(* IEC 61131-3 sources: SIMERLIFT/LOGICAD/SIMERLIFT/src_FBD/BCU/fbdBCU_bess (part 2) *)

  @G(1535) :
     @L(@VF(1532).o, @C(1530).CODE)
    ;
  @G(1536) :
     @L(@VF(1533).o, @C(1530).R)
    ;
  @G(257) :
     @L(@VF(165).o, @C(1).OVTHRES)
    ;
  @G(155) :
     @L(@VF(19).o, @C(1).BAUD)
    ;
  @G(252) :
     @L(@VF(167).o, @C(1).UVTHRES)
    ;
  @G(538) :
     @L(@VF(536).o, @C(1).M_ALL_R)
    ;
  @G(539) :
     @L(@VF(537).o, @C(1).M_AUX_R)
    ;
  @G(206) :
     @L(@VF(24).o, @C(1).N_CELLS)
    ;
  @G(208) :
     @L(@VF(636).o, @C(1).T_CELLS)
    ;
  @G(209) :
     @L(@VF(26).o, @C(1).CHSEL)
    ;
  @G(210) :
     @L(@VF(126).o, @C(1).BRD)
    ;
  @G(213) :
     @L(@VF(235).o, @C(1).CELL)
    ;
  @G(217) :
     @L(@VF(35).o, @C(1).CH)
    ;
  @G(446) :
     @L(@VF(445).o, @C(1).BALV)
    ;
  @G(13) :
     @L(@C(1).VAV, @VF(48).i)
    ;
  @G(11) :
     @L(@C(1).VMINCELL, @VF(30).i)
    ;
  @G(10) :
     @L(@C(1).VMAXCELL, @VF(12).i)
    ;
  @G(8) :
     @L(@C(1).MINCELLBRD, @VF(6).i)
    ;
  @G(3) :
     @L(@C(1).MAXCELLNUM, @VF(5).i)
    ;
  @G(2) :
     @L(@C(1).MAXCELLBRD, @VF(4).i)
    ;
  @G(9) :
     @L(@C(1).MINCELLNUM, @VF(7).i)
    ;
  @G(31) :
     @L(@C(1).VCELL, @VF(18).i)
    ;
  @G(256) :
     @L(@VF(201).o, @C(1).BALENB)
    ;
  @G(41) :
     @L(@C(1).TEMPCELL, @VF(25).i)
    ;
  @G(770) :
     @L(@C(1).VSTACK, @VF(29).i)
    ;
  @G(271) :
     @L(@VF(119).o, @C(1).NTCNOMT_KLV)
    ;
  @G(272) :
     @L(@VF(121).o, @C(1).NTCNOMR_OHM)
    ;
  @G(44) :
     @L(@C(1).BALREG, @VF(72).i)
    ;
  @G(45) :
     @L(@C(1).N_BRD, @VF(154).i)
    ;
  @G(55) :
     @L(@C(1).FAULT, @VF(372).i)
    ;
  @G(128) :
     @L(@C(1).ERR, @VF(654).i)
    ;
  @G(21) :
     @L(@VF(16).o, @C(15).R)
    ;
  @G(27) :
     @L(@VF(20).o, @C(15).CODE)
    ;
  @G(649) :
     @L(@CP(467), @CP(1326)),
     @L(@CP(640), @C(104).CAN_CH),
     @L(@CP(640), @CP(353)),
     @L(@CP(1326), @CP(640)),
     @L(@CP(1326), @C(1004).CAN_CH),
     @L(@VF(638).o, @CP(467)),
     @L(@CP(353), @C(83).CAN_CH),
     @L(@CP(467), @C(136).CAN_CH),
     @L(@CP(353), @C(84).CAN_CH)
    ;
  @G(189) :
     @L(@VF(188).o, @C(1004).CAN_ID)
    ;
  @G(1330) :
     @L(@VF(1120).o, @C(1004).Instant_Current)
    ;
  @G(1331) :
     @L(@VF(1124).o, @C(1004).Selected_BMU_Loc)
    ;
  @G(1332) :
     @L(@VF(1123).o, @C(1004).Selected_Cell_Loc)
    ;
  @G(1333) :
     @L(@VF(1128).o, @C(1004).Cell_Voltage)
    ;
  @G(1334) :
     @L(@VF(1147).o, @C(1004).Cell_Temp)
    ;
  @G(1335) :
     @L(@C(1004).CAN_Error, @VF(1325).i)
    ;
  @G(191) :
     @L(@VF(190).o, @C(104).CAN_ID)
    ;
  @G(1151) :
     @L(@VF(94).o, @C(104).Max_Volt_Cell_Loc)
    ;
  @G(1152) :
     @L(@VF(103).o, @C(104).Max_Volt_BMU_Loc)
    ;
  @G(1153) :
     @L(@VF(105).o, @C(104).Min_Volt_Cell_Loc)
    ;
  @G(1154) :
     @L(@VF(108).o, @C(104).Min_Volt_BMU_Loc)
    ;
  @G(1155) :
     @L(@VF(113).o, @C(104).Average_Cell_Voltage)
    ;
  @G(1156) :
     @L(@VF(114).o, @C(104).Max_Cell_Voltage)
    ;
  @G(1159) :
     @L(@C(104).CAN_Error, @VF(745).i)
    ;
  @G(1160) :
     @L(@VF(115).o, @C(104).Min_Cell_Voltage)
    ;
  @G(782) :
     @L(@C(778).DIV, @VF(779).i)
    ;
  @G(1525) :
     @L(@C(1520).DIV, @VF(1519).i)
    ;
  @G(783) :
     @L(@VF(781).o, @CP(1521)),
     @L(@CP(1521), @C(778).IN2),
     @L(@CP(1521), @C(1520).IN2),
     @L(@CP(1521), @C(1880).IN2),
     @L(@CP(1521), @C(43).IN2)
    ;
  @G(1524) :
     @L(@VF(523).o, @C(1520).IN1)
    ;
  @G(1885) :
     @L(@VF(524).o, @C(1880).IN1)
    ;
  @G(142) :
     @L(@C(466).Overall_Power_kWh, @VF(982).i)
    ;
  @G(717) :
     @L(@C(466).Current_Counter_Ah, @VF(678).i)
    ;
  @G(715) :
     @L(@C(466).Power_kWh, @VF(664).i)
    ;
  @G(713) :
     @L(@C(466).Temp, @VF(663).i)
    ;
  @G(528) :
     @L(@C(466).Voltage3_mV, @VF(525).i)
    ;
  @G(527) :
     @L(@C(466).Voltage2_mV, @VF(524).i)
    ;
  @G(526) :
     @L(@C(466).Voltage1_mV, @VF(523).i)
    ;
  @G(825) :
     @L(@VF(824).o, @C(800).ENB)
    ;
  @G(227) :
     @L(@VF(1526).o, @C(218).SoC)
    ;
  @G(228) :
     @L(@VF(1500).o, @C(218).SoH)
    ;
  @G(229) :
     @L(@VF(1498).o, @C(218).Voltage)
    ;
  @G(681) :
     @L(@VF(1490).o, @C(218).Current)
    ;
  @G(714) :
     @L(@VF(1492).o, @C(218).Temp)
    ;
  @G(752) :
     @L(@VF(1499).o, @C(218).Fault)
    ;
  @G(764) :
     @L(@VF(1389).o, @C(218).Cycle)
    ;
  @G(927) :
     @L(@VF(1390).o, @C(218).State)
    ;
  @G(1037) :
     @L(@VF(1391).o, @C(218).ID)
    ;
  @G(1039) :
     @L(@VF(1038).o, @C(218).CH)
    ;
  @G(1979) :
     @L(@VF(984).o, @C(1978).IN1)
    ;
  @G(1980) :
     @L(@VF(1977).o, @C(1978).IN2)
    ;
  @G(1986) :
     @L(@VF(1984).o, @C(1985).IN1)
    ;
  @G(1982) :
     @L(@C(1978).DIV, @C(1981).IN)
    ;
  @G(1991) :
     @L(@VF(1989).o, @C(1990).IN1)
    ;
  @G(1992) :
     @L(@C(1985).DIV, @C(1990).IN2)
    ;
  @G(1983) :
     @L(@C(1981).TO_USINT, @VF(986).i)
    ;
  @G(1994) :
     @L(@C(1990).SUB, @C(1993).IN)
    ;
  @G(1999) :
     @L(@VF(1998).o, @C(1993).MX)
    ;
  @G(2001) :
     @L(@VF(2000).o, @C(1993).MN)
    ;
  @G(1997) :
     @L(@C(1993).LIMIT, @C(1995).IN)
    ;
  @G(1996) :
     @L(@C(1995).TO_USINT, @VF(129).i)
    ;
  @G(107) :
     @L(@VF(40).o, @C(1).ENB)
    ;
  @G(1571) :
     @L(@VF(1569).o, @C(1580).IN2)
    ;
  @G(1572) :
     @L(@VF(1558).o, @CP(1579)),
     @L(@CP(1579), @C(364).IN1),
     @L(@CP(1579), @C(1580).IN1)
    ;
  @G(1573) :
     @L(@VF(1560).o, @CP(1584)),
     @L(@CP(1584), @C(404).IN1),
     @L(@CP(1584), @C(1582).IN1)
    ;
  @G(1561) :
     @L(@VF(1559).o, @C(1582).IN2)
    ;
  @G(1565) :
     @L(@C(364).GE, @C(161).IN)
    ;
  @G(1576) :
     @L(@VF(1575).o, @C(161).PT)
    ;
  @G(1566) :
     @L(@VF(1564).o, @C(234).PT)
    ;
  @G(1577) :
     @L(@C(404).LE, @C(234).IN)
    ;
  @G(1602) :
     @L(@C(1582).LE, @C(1583).IN)
    ;
  @G(1607) :
     @L(@VF(1591).o, @C(1583).PT)
    ;
  @G(1686) :
     @L(@C(279).GE, @C(921).IN)
    ;
  @G(1682) :
     @L(@VF(1659).o, @CP(1589)),
     @L(@CP(1589), @C(279).IN1),
     @L(@CP(1589), @C(920).IN1)
    ;
  @G(1600) :
     @L(@VF(1588).o, @C(1581).PT)
    ;
  @G(1599) :
     @L(@C(1580).GE, @C(1581).IN)
    ;
  @G(1679) :
     @L(@VF(1662).o, @CP(1590)),
     @L(@CP(1590), @C(276).IN1),
     @L(@CP(1590), @C(920).IN2)
    ;
  @G(1680) :
     @L(@C(276).SUB, @C(279).IN2)
    ;
  @G(1687) :
     @L(@VF(1665).o, @C(921).PT)
    ;
  @G(1676) :
     @L(@VF(1348).o, @C(276).IN2)
    ;
  @G(1690) :
     @L(@C(920).GE, @C(1060).IN)
    ;
  @G(1691) :
     @L(@VF(1668).o, @C(1060).PT)
    ;
  @G(1689) :
     @L(@C(919).LE, @C(1058).IN)
    ;
  @G(1598) :
     @L(@VF(1660).o, @CP(1664)),
     @L(@CP(1664), @C(919).IN1),
     @L(@CP(1664), @C(1073).IN1)
    ;
  @G(1563) :
     @L(@C(161).Q, @VF(1555).i)
    ;
  @G(1578) :
     @L(@C(234).Q, @VF(1556).i)
    ;
  @G(1604) :
     @L(@C(1583).Q, @VF(1594).i)
    ;
  @G(1692) :
     @L(@C(921).Q, @VF(1672).i)
    ;
  @G(1693) :
     @L(@C(1058).Q, @VF(1673).i)
    ;
  @G(1694) :
     @L(@C(1060).Q, @VF(1674).i)
    ;
  @G(1603) :
     @L(@C(1581).Q, @VF(1593).i)
    ;
  @G(1681) :
     @L(@C(277).ADD, @C(919).IN2)
    ;
  @G(1688) :
     @L(@VF(1666).o, @C(1058).PT)
    ;
  @G(1678) :
     @L(@VF(1661).o, @CP(1601)),
     @L(@CP(1601), @C(277).IN1),
     @L(@CP(1601), @C(1073).IN2)
    ;
  @G(1677) :
     @L(@VF(1663).o, @C(277).IN2)
    ;
  @G(1696) :
     @L(@C(1073).LE, @C(1347).IN)
    ;
  @G(1697) :
     @L(@C(1347).Q, @VF(1675).i)
    ;
  @G(1698) :
     @L(@VF(1671).o, @C(1347).PT)
    ;
  @G(1052) :
     @L(@VF(1056).o, @C(803).IN1)
    ;
  @G(1054) :
     @L(@C(803).LT, @C(997).I)
    ;
  @G(1820) :
     @L(@C(1819).OR, @VF(1670).i)
    ;
  @G(1821) :
     @L(@C(997).O, @C(1819).IN1)
    ;
  @G(1667) :
     @L(@VF(1050).o, @C(803).IN2)
    ;
  @G(1822) :
     @L(@C(1817).O, @C(1819).IN2)
    ;
  @G(1818) :
     @L(@C(1669).LT, @C(1817).I)
    ;
  @G(1703) :
     @L(@C(1684).GT, @C(1683).I)
    ;
  @G(1704) :
     @L(@VF(1685).o, @C(1684).IN1)
    ;
  @G(1823) :
     @L(@C(1683).O, @C(1706).IN1)
    ;
  @G(1824) :
     @L(@C(1706).OR, @VF(1699).i)
    ;
  @G(1705) :
     @L(@VF(1695).o, @C(1684).IN2)
    ;
  @G(1831) :
     @L(@C(1830).O, @C(1706).IN2)
    ;
  @G(1832) :
     @L(@C(1825).GT, @C(1830).I)
    ;
  @G(141) :
     @L(@VF(164).o, @C(972).IN)
    ;
  @G(791) :
     @L(@VF(124).o, @C(962).IN)
    ;
  @G(974) :
     @L(@C(972).TO_REAL, @C(971).IN2)
    ;
  @G(503) :
     @L(@VF(497).o, @C(502).IN2)
    ;
  @G(960) :
     @L(@C(958).MUL, @C(959).IN1)
    ;
  @G(976) :
     @L(@C(971).MUL, @C(975).IN1)
    ;
  @G(595) :
     @L(@C(502).MUL, @C(509).IN1)
    ;
  @G(967) :
     @L(@C(959).DIV, @VF(954).i)
    ;
  @G(969) :
     @L(@C(975).DIV, @VF(955).i)
    ;
  @G(687) :
     @L(@C(517).MUL, @C(336).IN1)
    ;
  @G(144) :
     @L(@C(509).DIV, @VF(506).i)
    ;
  @G(501) :
     @L(@C(336).DIV, @VF(278).i)
    ;
  @G(711) :
     @L(@VF(709).o, @C(517).IN2)
    ;
  @G(392) :
     @L(@VF(964).o, @C(887).IN2)
    ;
  @G(552) :
     @L(@VF(551).o, @C(544).IN1)
    ;
  @G(545) :
     @L(@C(887).GE, @C(542).IN1)
    ;
  @G(546) :
     @L(@C(544).GE, @C(542).IN2)
    ;
  @G(1716) :
     @L(@C(542).OR, @C(1702).IN1)
    ;
  @G(885) :
     @L(@VF(832).o, @C(544).IN2)
    ;
  @G(1712) :
     @L(@VF(1711).o, @C(548).PT)
    ;
  @G(1725) :
     @L(@C(1702).AND, @C(548).IN)
    ;
  @G(1710) :
     @L(@C(548).Q, @C(895).S1)
    ;
  @G(666) :
     @L(@C(895).Q1, @VF(68).i)
    ;
  @G(49) :
     @L(@C(979).PACK_ID, @VF(980).i)
    ;
  @G(50) :
     @L(@C(979).CAN_ID_10, @VF(993).i)
    ;
  @G(51) :
     @L(@C(979).CAN_ID_11, @VF(992).i)
    ;
  @G(52) :
     @L(@C(979).CAN_ID_12, @VF(988).i)
    ;
  @G(53) :
     @L(@C(979).CAN_ID_13, @VF(981).i)
    ;
  @G(54) :
     @L(@C(979).CAN_ID_14, @VF(994).i)
    ;
  @G(56) :
     @L(@C(979).CAN_ID_15, @VF(995).i)
    ;
  @G(57) :
     @L(@C(979).CAN_ID_16, @VF(996).i)
    ;
  @G(836) :
     @L(@C(125).chState, @VF(773).i)
    ;
  @G(841) :
     @L(@C(125).balance, @VF(772).i)
    ;
  @G(842) :
     @L(@C(125).complete, @VF(151).i)
    ;
  @G(813) :
     @L(@VF(499).o, @C(125).mainComplete)
    ;
  @G(162) :
     @L(@VF(440).o, @C(125).dmcc)
    ;
  @G(163) :
     @L(@VF(156).o, @C(125).battAmpr)
    ;
  @G(827) :
     @L(@VF(767).o, @C(125).balAmpr)
    ;
  @G(830) :
     @L(@VF(769).o, @C(125).maxCell)
    ;
  @G(835) :
     @L(@VF(1141).o, @C(125).minCell)
    ;
  @G(2007) :
     @L(@C(146).state, @VF(2006).i)
    ;
  @G(166) :
     @L(@VF(159).o, @C(146).chargeCompleted)
    ;
  @G(2003) :
     @L(@C(146).remainingWh, @CP(135)),
     @L(@CP(135), @VF(2002).i),
     @L(@CP(135), @C(816).IN1)
    ;
  @G(171) :
     @L(@VF(158).o, @C(146).instantWh)
    ;
  @G(802) :
     @L(@C(793).EQ, @C(125).chargeOn)
    ;
  @G(985) :
     @L(@C(933).TO_USINT, @VF(172).i)
    ;
  @G(794) :
     @L(@VF(792).o, @C(793).IN2)
    ;
  @G(801) :
     @L(@VF(160).o, @C(793).IN1)
    ;
  @G(818) :
     @L(@VF(814).o, @C(815).CLK)
    ;
  @G(438) :
     @L(@C(413).Balance_Enable, @VF(414).i)
    ;
  @G(67) :
     @L(@C(413).Ballance_Voltage, @VF(447).i)
    ;
  @G(473) :
     @L(@C(413).Measure_All, @VF(532).i)
    ;
  @G(490) :
     @L(@C(413).Measure_Aux, @VF(534).i)
    ;
  @G(498) :
     @L(@VF(66).o, @C(413).Max_Cell_Voltage)
    ;
  @G(529) :
     @L(@VF(465).o, @C(413).Min_Cell_Voltage)
    ;
  @G(531) :
     @L(@VF(470).o, @C(413).Avarage_Cell_Voltage)
    ;
  @G(533) :
     @L(@VF(495).o, @C(413).Balance_Threshold)
    ;
  @G(541) :
     @L(@VF(530).o, @C(413).Ballance_Interval)
    ;
  @G(540) :
     @L(@VF(492).o, @C(413).Charge_Status)
    ;
  @G(33) :
     @L(@VF(34).o, @C(32).numofBMU)
    ;
  @G(36) :
     @L(@VF(37).o, @C(32).cellMap)
    ;
  @G(38) :
     @L(@C(32).numofCell, @VF(28).i)
    ;
  @G(494) :
     @L(@C(324).Q, @VF(361).i)
    ;
  @G(450) :
     @L(@VF(325).o, @C(324).PT)
    ;
  @G(451) :
     @L(@C(322).O, @C(324).IN)
    ;
  @G(247) :
     @L(@C(243).NE, @C(322).I)
    ;
  @G(254) :
     @L(@VF(248).o, @C(243).IN1)
    ;
  @G(255) :
     @L(@VF(250).o, @C(243).IN2)
    ;
  @G(601) :
     @L(@C(405).Q, @VF(338).i)
    ;
  @G(839) :
     @L(@C(369).Q, @VF(339).i)
    ;
  @G(852) :
     @L(@C(368).Q, @VF(340).i)
    ;
  @G(727) :
     @L(@C(366).Q, @VF(337).i)
    ;
  @G(600) :
     @L(@VF(593).o, @C(405).PT)
    ;
  @G(718) :
     @L(@VF(602).o, @C(366).PT)
    ;
  @G(729) :
     @L(@VF(370).o, @C(368).PT)
    ;
  @G(730) :
     @L(@VF(371).o, @C(369).PT)
    ;
  @G(1049) :
     @L(@C(826).O, @C(369).IN)
    ;
  @G(1055) :
     @L(@C(728).O, @C(366).IN)
    ;
  @G(367) :
     @L(@VF(292).o, @C(405).IN)
    ;
  @G(283) :
     @L(@VF(261).o, @C(258).PT)
    ;
  @G(1835) :
     @L(@VF(262).o, @C(1813).IN2)
    ;
  @G(1051) :
     @L(@C(286).LE, @C(826).I)
    ;
  @G(1053) :
     @L(@C(288).GE, @C(728).I)
    ;
  @G(285) :
     @L(@C(258).Q, @VF(925).i)
    ;
  @G(1834) :
     @L(@VF(264).o, @C(1813).IN1)
    ;
  @G(1836) :
     @L(@C(1813).OR, @C(258).IN)
    ;
  @G(289) :
     @L(@VF(263).o, @C(1071).I)
    ;
  @G(918) :
     @L(@VF(677).o, @C(281).PT)
    ;
  @G(1837) :
     @L(@C(259).OR, @C(281).IN)
    ;
  @G(1839) :
     @L(@VF(1838).o, @C(259).IN2)
    ;
  @G(1840) :
     @L(@VF(268).o, @C(259).IN1)
    ;
  @G(403) :
     @L(@VF(398).o, @C(393).PT)
    ;
  @G(396) :
     @L(@C(393).Q, @VF(332).i)
    ;
  @G(1059) :
     @L(@C(394).O, @C(393).IN)
    ;
  @G(293) :
     @L(@VF(266).o, @C(394).I)
    ;
  @G(294) :
     @L(@VF(273).o, @C(288).IN1)
    ;
  @G(309) :
     @L(@VF(274).o, @C(286).IN1)
    ;
  @G(311) :
     @L(@VF(280).o, @C(286).IN2)
    ;
  @G(312) :
     @L(@VF(282).o, @C(288).IN2)
    ;
  @G(298) :
     @L(@C(1071).O, @C(297).IN)
    ;
  @G(299) :
     @L(@C(297).Q, @VF(334).i)
    ;
  @G(301) :
     @L(@VF(300).o, @C(297).PT)
    ;
  @G(348) :
     @L(@C(1).MAXTEMPBRD, @VF(1102).i)
    ;
  @G(349) :
     @L(@C(1).MAXTEMPCELL, @VF(1103).i)
    ;
  @G(350) :
     @L(@C(1).MINTEMPBRD, @VF(1101).i)
    ;
  @G(351) :
     @L(@C(1).MINTEMPCELL, @VF(1100).i)
    ;
  @G(400) :
     @L(@CP(399), @C(388).CAN_CH),
     @L(@CP(399), @C(395).CAN_CH),
     @L(@VF(389).o, @CP(399))
    ;
  @G(401) :
     @L(@VF(390).o, @C(388).CAN_ID)
    ;
  @G(418) :
     @L(@C(415).TO_UINT, @C(388).IN_1)
    ;
  @G(426) :
     @L(@C(419).TO_UINT, @C(388).IN_2)
    ;
  @G(430) :
     @L(@C(420).TO_UINT, @C(388).IN_3)
    ;
  @G(431) :
     @L(@C(421).TO_UINT, @C(388).IN_4)
    ;
  @G(432) :
     @L(@VF(391).o, @C(395).CAN_ID)
    ;
  @G(433) :
     @L(@C(422).TO_UINT, @C(395).IN_1)
    ;
  @G(406) :
     @L(@C(423).TO_UINT, @C(395).IN_2)
    ;
  @G(777) :
     @L(@C(424).TO_UINT, @C(395).IN_3)
    ;
  @G(407) :
     @L(@C(425).TO_UINT, @C(395).IN_4)
    ;
  @G(472) :
     @L(@C(962).TO_REAL, @C(958).IN2)
    ;
  @G(482) :
     @L(@VF(968).o, @C(959).IN2)
    ;
  @G(484) :
     @L(@VF(483).o, @C(975).IN2)
    ;
  @G(488) :
     @L(@VF(485).o, @C(509).IN2)
    ;
  @G(513) :
     @L(@VF(493).o, @C(336).IN2)
    ;
  @G(608) :
     @L(@VF(578).o, @C(570).Fault_07)
    ;
  @G(609) :
     @L(@VF(577).o, @C(570).Fault_06)
    ;
  @G(611) :
     @L(@VF(928).o, @C(570).Fault_05)
    ;
  @G(612) :
     @L(@VF(572).o, @C(570).Fault_04)
    ;
  @G(613) :
     @L(@VF(929).o, @C(570).Fault_03)
    ;
  @G(618) :
     @L(@VF(571).o, @C(570).Fault_02)
    ;
  @G(620) :
     @L(@VF(576).o, @C(570).Fault_01)
    ;
  @G(622) :
     @L(@VF(575).o, @C(570).Fault_00)
    ;
  @G(624) :
     @L(@VF(573).o, @C(570).CAN_CH)
    ;
  @G(629) :
     @L(@VF(574).o, @C(570).CAN_ID)
    ;
  @G(637) :
     @L(@VF(579).o, @C(570).Fault_08)
    ;
  @G(639) :
     @L(@VF(583).o, @C(570).Fault_09)
    ;
  @G(645) :
     @L(@VF(589).o, @C(570).Fault_12)
    ;
  @G(646) :
     @L(@VF(590).o, @C(570).Fault_13)
    ;
  @G(647) :
     @L(@VF(591).o, @C(570).Fault_14)
    ;
  @G(648) :
     @L(@VF(594).o, @C(570).Fault_15)
    ;
  @G(661) :
     @L(@VF(660).o, @C(570).Fault_16)
    ;
  @G(863) :
     @L(@C(570).GUI_Fault, @VF(862).i)
    ;
  @G(737) :
     @L(@VF(736).o, @C(570).Fault_33)
    ;
  @G(680) :
     @L(@VF(679).o, @C(570).Fault_Byte_5)
    ;
  @G(650) :
     @L(@VF(596).o, @C(570).Fault_Byte_6_7)
    ;
  @G(598) :
     @L(@VF(98).o, @C(97).VAL)
    ;
  @G(599) :
     @L(@VF(101).o, @C(81).VAL)
    ;
  @G(603) :
     @L(@VF(100).o, @C(81).PORT)
    ;
  @G(604) :
     @L(@VF(99).o, @C(81).PIN)
    ;
  @G(614) :
     @L(@VF(462).o, @C(97).PIN)
    ;
  @G(615) :
     @L(@VF(463).o, @C(97).PORT)
    ;
  @G(199) :
     @L(@C(281).Q, @VF(924).i)
    ;
  @G(674) :
     @L(@VF(653).o, @C(887).IN1)
    ;
  @G(476) :
     @L(@VF(693).o, @CP(477)),
     @L(@CP(477), @C(958).IN1),
     @L(@CP(477), @C(971).IN1),
     @L(@CP(477), @C(502).IN1),
     @L(@CP(477), @C(517).IN1),
     @L(@CP(477), @C(1353).IN1),
     @L(@CP(477), @C(479).IN1)
    ;
  @G(559) :
     @L(@C(466).CAN_Error, @VF(478).i)
    ;
  @G(795) :
     @L(@C(763).Q, @CP(787)),
     @L(@CP(787), @C(762).CU),
     @L(@CP(787), @C(763).R)
    ;
  @G(805) :
     @L(@C(762).CV, @C(765).IN)
    ;
  @G(806) :
     @L(@C(763).CV, @C(766).IN)
    ;
  @G(807) :
     @L(@C(765).TO_USINT, @VF(785).i)
    ;
  @G(808) :
     @L(@C(766).TO_USINT, @VF(786).i)
    ;
  @G(788) :
     @L(@C(706).OUT, @CP(1914)),
     @L(@CP(1914), @C(763).CU),
     @L(@CP(1914), @VF(1913).i)
    ;
  @G(789) :
     @L(@VF(768).o, @C(706).IN)
    ;
  @G(790) :
     @L(@VF(774).o, @C(706).PER)
    ;
  @G(1221) :
     @L(@VF(584).o, @C(778).IN1)
    ;
  @G(1357) :
     @L(@VF(1354).o, @C(1352).IN2)
    ;
  @G(1359) :
     @L(@C(1353).MUL, @C(1352).IN1)
    ;
  @G(1360) :
     @L(@C(1352).DIV, @VF(1355).i)
    ;
  @G(1358) :
     @L(@VF(1356).o, @C(1353).IN2)
    ;
  @G(1400) :
     @L(@C(570).sum, @VF(1399).i)
    ;
  @G(1700) :
     @L(@CP(1714), @C(1658).IN1),
     @L(@CP(1714), @C(1713).IN1),
     @L(@VF(335).o, @CP(1714))
    ;
  @G(1708) :
     @L(@VF(1701).o, @C(1658).IN2)
    ;
  @G(1717) :
     @L(@VF(1715).o, @C(1713).IN2)
    ;
  @G(1720) :
     @L(@C(1658).EQ, @CP(138)),
     @L(@CP(138), @C(1719).IN1),
     @L(@CP(138), @VF(137).i)
    ;
  @G(1721) :
     @L(@C(1713).EQ, @CP(365)),
     @L(@CP(365), @C(1719).IN2),
     @L(@CP(365), @VF(362).i)
    ;
  @G(1856) :
     @L(@VF(1767).o, @C(1762).IN2)
    ;
  @G(1860) :
     @L(@C(1762).DIV, @C(1771).IN)
    ;
  @G(1861) :
     @L(@C(1770).DIV, @C(1772).IN)
    ;
  @G(1899) :
     @L(@VF(1814).o, @C(1789).IN)
    ;
  @G(1901) :
     @L(@C(1789).TO_UINT, @VF(1826).i)
    ;
  @G(1902) :
     @L(@C(1788).TO_UINT, @VF(1827).i)
    ;
  @G(1424) :
     @L(@VF(1420).o, @C(1419).PORT)
    ;
  @G(1423) :
     @L(@VF(1421).o, @C(1419).PIN)
    ;
  @G(1425) :
     @L(@VF(1422).o, @C(1419).VAL)
    ;
  @G(1414) :
     @L(@VF(1346).o, @C(1344).ADC)
    ;
  @G(1415) :
     @L(@VF(1349).o, @C(1344).GRP)
    ;
  @G(1416) :
     @L(@VF(1351).o, @C(1344).CH)
    ;
  @G(454) :
     @L(@VF(676).o, @C(1004).Total_Voltage)
    ;
  @G(207) :
     @L(@VF(79).o, @C(74).IN2)
    ;
  @G(211) :
     @L(@VF(78).o, @C(74).IN1)
    ;
  @G(623) :
     @L(@C(74).MUL, @C(73).IN)
    ;
  @G(222) :
     @L(@VF(80).o, @C(74).IN3)
    ;
  @G(304) :
     @L(@VF(102).o, @C(74).IN4)
    ;
  @G(305) :
     @L(@C(73).TO_REAL, @C(75).IN1)
    ;
  @G(306) :
     @L(@VF(96).o, @C(75).IN2)
    ;
  @G(1368) :
     @L(@VF(177).o, @C(1367).IN1)
    ;
  @G(1448) :
     @L(@C(1367).MUL, @CP(194)),
     @L(@CP(194), @VF(179).i),
     @L(@CP(194), @C(77).IN1)
    ;
  @G(2076) :
     @L(@VF(2075).o, @C(2073).IN2)
    ;
  @G(354) :
     @L(@C(77).MUL, @VF(186).i)
    ;
  @G(2078) :
     @L(@C(2073).MUL, @C(2077).IN1)
    ;
  @G(2080) :
     @L(@VF(2079).o, @C(2077).IN2)
    ;
  @G(2082) :
     @L(@C(2077).DIV, @VF(2081).i)
    ;
  @G(1454) :
     @L(@VF(1452).o, @C(77).IN2)
    ;
  @G(307) :
     @L(@C(75).DIV, @VF(183).i)
    ;
  @G(455) :
     @L(@VF(183).o, @C(2073).IN1)
    ;
  @G(352) :
     @L(@VF(187).o, @C(1367).IN2)
    ;
  @G(486) :
     @L(@VF(173).o, @C(146).capacityWh)
    ;
  @G(123) :
     @L(@C(816).DIV, @VF(118).i)
    ;
  @G(131) :
     @L(@VF(120).o, @C(816).IN2)
    ;
  @G(508) :
     @L(@C(505).O, @C(507).IN)
    ;
  @G(512) :
     @L(@C(507).Q, @VF(511).i)
    ;
  @G(580) :
     @L(@VF(547).o, @C(507).PT)
    ;
  @G(592) :
     @L(@VF(504).o, @C(510).IN)
    ;
  @G(597) :
     @L(@C(510).NOT, @C(505).I)
    ;
  @G(631) :
     @L(@VF(1815).o, @C(1788).IN)
    ;
  @G(634) :
     @L(@C(125).chargeAmpr, @VF(628).i)
    ;
  @G(643) :
     @L(@VF(635).o, @C(218).Humidity)
    ;
  @G(809) :
     @L(@VF(799).o, @C(762).PV)
    ;
  @G(377) :
     @L(@VF(170).o, @C(1825).IN2)
    ;
  @G(402) :
     @L(@VF(458).o, @C(1669).IN2)
    ;
  @G(630) :
     @L(@VF(521).o, @C(459).IN2)
    ;
  @G(632) :
     @L(@C(459).DIV, @VF(522).i)
    ;
  @G(633) :
     @L(@C(479).MUL, @C(459).IN1)
    ;
  @G(691) :
     @L(@VF(586).o, @C(479).IN2)
    ;
  @G(698) :
     @L(@VF(1177).o, @C(1161).CODE)
    ;
  @G(701) :
     @L(@VF(1179).o, @C(1161).R)
    ;
  @G(702) :
     @L(@VF(1541).o, @C(1539).CODE)
    ;
  @G(784) :
     @L(@VF(1542).o, @C(1539).R)
    ;
  @G(845) :
     @L(@C(1161).VAL, @C(1169).IN)
    ;
  @G(848) :
     @L(@C(1169).TO_UINT, @C(1184).IN1)
    ;
  @G(856) :
     @L(@VF(1197).o, @C(1184).IN2)
    ;
  @G(879) :
     @L(@C(1538).TO_UINT, @C(1194).IN1)
    ;
  @G(888) :
     @L(@VF(1199).o, @C(1194).IN2)
    ;
  @G(910) :
     @L(@C(1539).VAL, @C(1538).IN)
    ;
  @G(922) :
     @L(@C(1194).MIN, @VF(912).i)
    ;
  @G(941) :
     @L(@VF(936).o, @C(932).IN1)
    ;
  @G(943) :
     @L(@VF(937).o, @C(932).IN2)
    ;
  @G(1214) :
     @L(@VF(1212).o, @C(1213).IN)
    ;
  @G(1216) :
     @L(@C(1213).TO_DWORD, @CP(1223)),
     @L(@CP(1223), @C(1215).IN1),
     @L(@CP(1223), @C(934).IN1),
     @L(@CP(1223), @C(1229).IN1)
    ;
  @G(1220) :
     @L(@VF(1218).o, @C(1215).IN2)
    ;
  @G(1225) :
     @L(@VF(1224).o, @C(934).IN2)
    ;
  @G(948) :
     @L(@VF(938).o, @C(935).D)
    ;
  @G(949) :
     @L(@C(932).NE, @C(935).I)
    ;
  @G(1228) :
     @L(@C(1229).AND, @C(1227).IN)
    ;
  @G(1238) :
     @L(@C(934).AND, @C(1233).IN)
    ;
  @G(1241) :
     @L(@C(1215).AND, @C(1239).IN)
    ;
  @G(1232) :
     @L(@VF(1230).o, @C(1229).IN2)
    ;
  @G(1244) :
     @L(@C(1227).TO_BOOL, @C(1243).IN3)
    ;
  @G(1942) :
     @L(@C(1233).TO_BOOL, @C(1243).IN2)
    ;
  @G(1943) :
     @L(@C(1239).TO_BOOL, @C(1243).IN1)
    ;
  @G(1944) :
     @L(@C(1243).OR, @C(1242).I)
    ;
  @G(1951) :
     @L(@VF(1950).o, @C(1242).D)
    ;
  @G(950) :
     @L(@C(935).O, @C(1226).IN1)
    ;
  @G(1945) :
     @L(@C(1242).O, @C(1226).IN2)
    ;
  @G(1245) :
     @L(@C(1226).OR, @VF(939).i)
    ;
  @G(720) :
     @L(@VF(553).o, @C(364).IN2)
    ;
  @G(732) :
     @L(@VF(658).o, @C(404).IN2)
    ;
  @G(417) :
     @L(@VF(822).o, @CP(823)),
     @L(@CP(823), @C(800).CH),
     @L(@CP(823), @C(466).CAN_CH)
    ;
  @G(881) :
     @L(@C(869).TO_UINT, @C(868).IN1)
    ;
  @G(882) :
     @L(@VF(872).o, @C(868).IN2)
    ;
  @G(883) :
     @L(@C(870).VAL, @C(869).IN)
    ;
  @G(884) :
     @L(@VF(875).o, @C(870).CODE)
    ;
  @G(891) :
     @L(@VF(876).o, @C(870).R)
    ;
  @G(871) :
     @L(@C(868).MIN, @VF(893).i)
    ;
  @G(902) :
     @L(@VF(900).o, @C(897).IN2)
    ;
  @G(911) :
     @L(@C(897).GE, @C(903).I)
    ;
  @G(914) :
     @L(@VF(913).o, @C(903).D)
    ;
  @G(916) :
     @L(@C(903).O, @VF(915).i)
    ;
  @G(963) :
     @L(@C(917).GE, @C(961).I)
    ;
  @G(966) :
     @L(@VF(965).o, @C(961).D)
    ;
  @G(973) :
     @L(@C(961).O, @VF(970).i)
    ;
  @G(978) :
     @L(@VF(977).o, @C(570).Fault_20)
    ;
  @G(1099) :
     @L(@VF(1095).o, @C(1093).PT)
    ;
  @G(1104) :
     @L(@VF(1096).o, @C(1092).IN2)
    ;
  @G(1105) :
     @L(@C(1093).Q, @VF(1098).i)
    ;
  @G(1106) :
     @L(@C(1094).O, @C(1093).IN)
    ;
  @G(1107) :
     @L(@C(1092).NE, @C(1094).I)
    ;
  @G(1108) :
     @L(@VF(1097).o, @C(1092).IN1)
    ;
  @G(1117) :
     @L(@VF(1112).o, @C(1110).PT)
    ;
  @G(1119) :
     @L(@VF(1113).o, @C(1109).IN2)
    ;
  @G(1121) :
     @L(@C(1110).Q, @VF(1116).i)
    ;
  @G(1122) :
     @L(@C(1111).O, @C(1110).IN)
    ;
  @G(1125) :
     @L(@C(1109).NE, @C(1111).I)
    ;
  @G(1126) :
     @L(@VF(1114).o, @C(1109).IN1)
    ;
  @G(1260) :
     @L(@C(1258).ABS, @C(1259).IN1)
    ;
  @G(1261) :
     @L(@VF(182).o, @C(1258).IN)
    ;
  @G(1263) :
     @L(@VF(1262).o, @C(1259).IN2)
    ;
  @G(181) :
     @L(@VF(180).o, @C(570).Fault_11)
    ;
  @G(185) :
     @L(@VF(184).o, @C(570).Fault_10)
    ;
  @G(321) :
     @L(@VF(76).o, @C(246).IN1)
    ;
  @G(333) :
     @L(@VF(331).o, @C(327).D)
    ;
  @G(342) :
     @L(@VF(655).o, @C(341).IN1)
    ;
  @G(907) :
     @L(@C(328).AND, @C(327).I)
    ;
  @G(1042) :
     @L(@C(341).LT, @C(328).IN2)
    ;
  @G(326) :
     @L(@VF(323).o, @C(246).IN2)
    ;
  @G(1057) :
     @L(@C(327).O, @C(329).S1)
    ;
  @G(1061) :
     @L(@C(329).Q1, @VF(1118).i)
    ;
  @G(1320) :
     @L(@C(246).LT, @C(906).IN1)
    ;
  @G(1321) :
     @L(@C(906).OR, @C(328).IN1)
    ;
  @G(1327) :
     @L(@C(1324).LT, @C(906).IN2)
    ;
  @G(1337) :
     @L(@VF(1322).o, @C(1324).IN1)
    ;
  @G(1339) :
     @L(@VF(1338).o, @C(1324).IN2)
    ;
  @G(443) :
     @L(@VF(1127).o, @C(570).Fault_21)
    ;
  @G(1404) :
     @L(@VF(1048).o, @C(570).Fault_22)
    ;
  @G(1272) :
     @L(@C(1719).OR, @VF(1718).i)
    ;
  @G(60) :
     @L(@C(1530).VAL, @C(23).IN)
    ;
  @G(62) :
     @L(@C(15).VAL, @C(61).IN)
    ;
  @G(1136) :
     @L(@C(1132).VAL, @C(998).IN)
    ;
  @G(1137) :
     @L(@VF(1133).o, @C(1132).CODE)
    ;
  @G(1158) :
     @L(@VF(1134).o, @C(1132).R)
    ;
  @G(1395) :
     @L(@C(998).TO_UINT, @VF(1394).i)
    ;
  @G(1408) :
     @L(@VF(1405).o, @C(1402).R)
    ;
  @G(1409) :
     @L(@C(1402).VAL, @C(1401).IN)
    ;
  @G(1411) :
     @L(@VF(1406).o, @C(1402).CODE)
    ;
  @G(1436) :
     @L(@VF(1429).o, @C(1428).R)
    ;
  @G(1437) :
     @L(@C(1428).VAL, @C(1426).IN)
    ;
  @G(1464) :
     @L(@VF(1430).o, @C(1428).CODE)
    ;
  @G(1472) :
     @L(@VF(1469).o, @C(1468).R)
    ;
  @G(1473) :
     @L(@C(1468).VAL, @C(1466).IN)
    ;
  @G(1474) :
     @L(@VF(1470).o, @C(1468).CODE)
    ;
  @G(1482) :
     @L(@VF(1479).o, @C(1478).R)
    ;
  @G(1483) :
     @L(@C(1478).VAL, @C(1477).IN)
    ;
  @G(1484) :
     @L(@VF(1480).o, @C(1478).CODE)
    ;
  @G(1493) :
     @L(@VF(1488).o, @C(1487).R)
    ;
  @G(1494) :
     @L(@C(1487).VAL, @C(1486).IN)
    ;
  @G(1495) :
     @L(@VF(1489).o, @C(1487).CODE)
    ;
  @G(1505) :
     @L(@VF(1502).o, @C(1501).R)
    ;
  @G(1506) :
     @L(@C(1501).VAL, @C(1497).IN)
    ;
  @G(1507) :
     @L(@VF(1503).o, @C(1501).CODE)
    ;
  @G(1413) :
     @L(@C(1401).TO_UINT, @VF(1407).i)
    ;
  @G(1465) :
     @L(@C(1426).TO_UINT, @VF(1431).i)
    ;
  @G(1475) :
     @L(@C(1466).TO_UINT, @VF(1471).i)
    ;
  @G(1485) :
     @L(@C(1477).TO_UINT, @VF(1481).i)
    ;
  @G(1496) :
     @L(@C(1486).TO_UINT, @VF(1491).i)
    ;
  @G(1508) :
     @L(@C(1497).TO_UINT, @VF(1504).i)
    ;
  @G(1523) :
     @L(@C(1510).VAL, @C(1509).IN)
    ;
  @G(1527) :
     @L(@VF(1512).o, @C(1510).R)
    ;
  @G(1531) :
     @L(@VF(1513).o, @C(1510).CODE)
    ;
  @G(1544) :
     @L(@C(1537).VAL, @C(1534).IN)
    ;
  @G(1545) :
     @L(@VF(1540).o, @C(1537).R)
    ;
  @G(1546) :
     @L(@VF(1543).o, @C(1537).CODE)
    ;
  @G(1548) :
     @L(@C(1509).TO_UINT, @VF(1547).i)
    ;
  @G(1550) :
     @L(@C(1534).TO_UINT, @VF(1549).i)
    ;
  @G(1557) :
     @L(@VF(1552).o, @C(1551).CODE)
    ;
  @G(1562) :
     @L(@VF(1554).o, @C(1551).R)
    ;
  @G(1568) :
     @L(@C(1551).VAL, @C(1567).IN)
    ;
  @G(1587) :
     @L(@C(1570).VAL, @C(1574).IN)
    ;
  @G(1592) :
     @L(@VF(1585).o, @C(1570).CODE)
    ;
  @G(1595) :
     @L(@VF(1586).o, @C(1570).R)
    ;
  @G(1597) :
     @L(@C(1567).TO_UINT, @VF(1596).i)
    ;
  @G(1606) :
     @L(@C(1574).TO_UINT, @VF(1605).i)
    ;
  @G(1611) :
     @L(@VF(1609).o, @C(1608).R)
    ;
  @G(1612) :
     @L(@VF(1610).o, @C(1608).CODE)
    ;
  @G(1614) :
     @L(@C(1608).VAL, @C(1613).IN)
    ;
  @G(1619) :
     @L(@C(1615).VAL, @C(1616).IN)
    ;
  @G(1620) :
     @L(@VF(1617).o, @C(1615).R)
    ;
  @G(1621) :
     @L(@VF(1618).o, @C(1615).CODE)
    ;
  @G(1626) :
     @L(@C(1622).VAL, @C(1623).IN)
    ;
  @G(1627) :
     @L(@VF(1624).o, @C(1622).R)
    ;
  @G(1628) :
     @L(@VF(1625).o, @C(1622).CODE)
    ;
  @G(1633) :
     @L(@C(1629).VAL, @C(1630).IN)
    ;
  @G(1634) :
     @L(@VF(1631).o, @C(1629).R)
    ;
  @G(1635) :
     @L(@VF(1632).o, @C(1629).CODE)
    ;
  @G(1724) :
     @L(@C(1613).TO_REAL, @VF(1723).i)
    ;
  @G(1726) :
     @L(@C(1616).TO_REAL, @VF(1722).i)
    ;
  @G(1727) :
     @L(@C(1623).TO_REAL, @VF(1636).i)
    ;
  @G(1728) :
     @L(@C(1630).TO_REAL, @VF(1637).i)
    ;
  @G(1734) :
     @L(@VF(1732).o, @C(1729).CODE)
    ;
  @G(1735) :
     @L(@VF(1733).o, @C(1729).R)
    ;
  @G(1736) :
     @L(@C(1729).VAL, @C(1731).IN)
    ;
  @G(1738) :
     @L(@C(1731).TO_UINT, @VF(1737).i)
    ;
  @G(1748) :
     @L(@C(1739).VAL, @C(1745).IN)
    ;
  @G(1749) :
     @L(@VF(1746).o, @C(1739).CODE)
    ;
  @G(1750) :
     @L(@VF(1747).o, @C(1739).R)
    ;
  @G(1753) :
     @L(@C(1745).TO_UINT, @VF(1752).i)
    ;
  @G(1877) :
     @L(@VF(1758).o, @C(1755).CODE)
    ;
  @G(1900) :
     @L(@VF(1757).o, @C(1755).R)
    ;
  @G(1756) :
     @L(@C(1755).VAL, @VF(1754).i)
    ;
  @G(1906) :
     @L(@VF(1904).o, @C(1903).CODE)
    ;
  @G(1907) :
     @L(@C(1903).VAL, @C(1799).IN)
    ;
  @G(1908) :
     @L(@VF(1905).o, @C(1903).R)
    ;
  @G(1910) :
     @L(@C(1799).TO_UINT, @VF(1909).i)
    ;
  @G(1912) :
     @L(@VF(1911).o, @C(1985).IN2)
    ;
  @G(2004) :
     @L(@VF(1987).o, @C(570).Fault_25)
    ;
  @G(2005) :
     @L(@VF(1988).o, @C(570).Fault_26)
    ;
  @G(2017) :
     @L(@VF(2016).o, @C(2011).IN5)
    ;
  @G(2018) :
     @L(@VF(2015).o, @C(2011).IN4)
    ;
  @G(2019) :
     @L(@VF(2014).o, @C(2011).IN3)
    ;
  @G(2020) :
     @L(@VF(2013).o, @C(2011).IN2)
    ;
  @G(2021) :
     @L(@VF(2012).o, @C(2011).IN1)
    ;
  @G(2022) :
     @L(@C(2011).OR, @VF(2010).i)
    ;
  @G(2042) :
     @L(@VF(2033).o, @C(2030).IN4)
    ;
  @G(2043) :
     @L(@VF(2031).o, @C(2030).IN2)
    ;
  @G(2044) :
     @L(@VF(2032).o, @C(2030).IN1)
    ;
  @G(2045) :
     @L(@VF(2034).o, @C(2030).IN3)
    ;
  @G(2046) :
     @L(@VF(2035).o, @C(2030).IN5)
    ;
  @G(2047) :
     @L(@VF(2036).o, @C(2030).IN6)
    ;
  @G(2050) :
     @L(@VF(2039).o, @C(2030).IN9)
    ;
  @G(2051) :
     @L(@VF(2040).o, @C(2030).IN10)
    ;
  @G(2052) :
     @L(@VF(2041).o, @C(2030).IN11)
    ;
  @G(2025) :
     @L(@C(2030).OR, @VF(2024).i)
    ;
  @G(2053) :
     @L(@VF(2023).o, @C(2030).IN12)
    ;
  @G(2048) :
     @L(@VF(2037).o, @C(2030).IN7)
    ;
  @G(2049) :
     @L(@VF(2038).o, @C(2030).IN8)
    ;
  @G(2055) :
     @L(@VF(2054).o, @C(2030).IN13)
    ;
  @G(2068) :
     @L(@VF(2058).o, @C(2056).IN6)
    ;
  @G(2069) :
     @L(@VF(2062).o, @C(2056).IN5)
    ;
  @G(2070) :
     @L(@VF(2060).o, @C(2056).IN4)
    ;
  @G(2071) :
     @L(@VF(2057).o, @C(2056).IN2)
    ;
  @G(2072) :
     @L(@VF(2059).o, @C(2056).IN1)
    ;
  @G(2074) :
     @L(@VF(2064).o, @C(2056).IN7)
    ;
  @G(2083) :
     @L(@VF(2063).o, @C(2056).IN8)
    ;
  @G(2084) :
     @L(@VF(2061).o, @C(2056).IN3)
    ;
  @G(2085) :
     @L(@VF(2065).o, @C(2056).IN9)
    ;
  @G(197) :
     @L(@C(1184).MIN, @VF(65).i)
    ;
  @G(2158) :
     @L(@C(2152).Q, @VF(2155).i)
    ;
  @G(2159) :
     @L(@C(2153).O, @C(2152).IN)
    ;
  @G(2160) :
     @L(@VF(2156).o, @C(2152).PT)
    ;
  @G(2161) :
     @L(@C(2154).NOT, @C(2153).I)
    ;
  @G(2162) :
     @L(@VF(2157).o, @C(2154).IN)
    ;
  @G(174) :
     @L(@VF(1237).o, @CP(176)),
     @L(@CP(176), @C(1669).IN1),
     @L(@CP(176), @C(1825).IN1)
    ;
  @G(2173) :
     @L(@C(2056).OR, @VF(2088).i)
    ;
  @G(287) :
     @L(@VF(71).o, @C(422).IN)
    ;
  @G(946) :
     @L(@VF(685).o, @C(423).IN)
    ;
  @G(2166) :
     @L(@VF(2116).o, @C(424).IN)
    ;
  @G(2178) :
     @L(@VF(2175).o, @C(2168).CODE)
    ;
  @G(2180) :
     @L(@VF(2176).o, @C(2168).R)
    ;
  @G(2177) :
     @L(@C(2168).VAL, @C(2174).IN)
    ;
  @G(2181) :
     @L(@C(2174).TO_UDINT, @VF(2179).i)
    ;
  @G(2205) :
     @L(@C(2202).VAL, @C(2201).IN)
    ;
  @G(2206) :
     @L(@VF(2203).o, @C(2202).CODE)
    ;
  @G(2207) :
     @L(@VF(2204).o, @C(2202).R)
    ;
  @G(2209) :
     @L(@C(2201).TO_UDINT, @VF(2208).i)
    ;
  @G(2212) :
     @L(@C(265).TO_REAL, @C(1).NTCBETA)
    ;
  @G(2213) :
     @L(@VF(117).o, @C(265).IN)
    ;
  @G(2087) :
     @L(@VF(2095).o, @C(2056).IN12)
    ;
  @G(2094) :
     @L(@VF(2090).o, @C(2056).IN11)
    ;
  @G(2247) :
     @L(@VF(2242).o, @C(2214).CODE)
    ;
  @G(2248) :
     @L(@VF(2243).o, @C(2214).R)
    ;
  @G(2244) :
     @L(@C(2214).VAL, @C(2096).IN)
    ;
  @G(2245) :
     @L(@C(2096).TO_UINT, @VF(2237).i)
    ;
  @G(956) :
     @L(@VF(953).o, @C(917).IN2)
    ;
  @G(2252) :
     @L(@VF(880).o, @C(2251).IN)
    ;
  @G(899) :
     @L(@C(2251).ABS, @CP(957)),
     @L(@CP(957), @C(897).IN1),
     @L(@CP(957), @C(917).IN1)
    ;
  @G(554) :
     @L(@VF(106).o, @C(2056).IN13)
    ;
  @G(675) :
     @L(@VF(616).o, @C(2030).IN14)
    ;
  @G(290) :
     @L(@VF(267).o, @C(368).IN)
    ;
  @G(317) :
     @L(@VF(109).o, @C(415).IN)
    ;
  @G(320) :
     @L(@VF(314).o, @C(419).IN)
    ;
  @G(439) :
     @L(@VF(192).o, @C(420).IN)
    ;
  @G(461) :
     @L(@VF(110).o, @C(421).IN)
    ;
  @G(1254) :
     @L(@VF(940).o, @C(753).IN2)
    ;
  @G(1255) :
     @L(@VF(1001).o, @C(755).IN2)
    ;
  @G(1256) :
     @L(@C(753).LT, @C(854).I)
    ;
  @G(1257) :
     @L(@VF(1251).o, @C(854).D)
    ;
  @G(1868) :
     @L(@VF(1209).o, @C(858).D)
    ;
  @G(1897) :
     @L(@C(755).GT, @C(858).I)
    ;
  @G(2254) :
     @L(@C(878).Q1, @VF(1253).i)
    ;
  @G(2271) :
     @L(@C(2255).MUX_USINT, @VF(2258).i)
    ;
  @G(2273) :
     @L(@C(2256).Battey_State_BCU_00, @C(2255).IN0)
    ;
  @G(2274) :
     @L(@C(2256).Battey_State_BCU_01, @C(2255).IN1)
    ;
  @G(2275) :
     @L(@C(2256).Battey_State_BCU_02, @C(2255).IN2)
    ;
  @G(2276) :
     @L(@C(2256).Battey_State_BCU_03, @C(2255).IN3)
    ;
  @G(2277) :
     @L(@C(2256).IMDCtrl_BCU0, @VF(2263).i)
    ;
  @G(2279) :
     @L(@C(2256).CAN_Error, @VF(2262).i)
    ;
  @G(2286) :
     @L(@CP(2269), @C(2256).CAN_CH),
     @L(@VF(2267).o, @CP(2269)),
     @L(@CP(2269), @C(90).CAN_CH)
    ;
  @G(2288) :
     @L(@VF(2266).o, @C(2256).CAN_ID)
    ;
  @G(86) :
     @L(@VF(82).o, @CP(88)),
     @L(@CP(88), @C(753).IN1),
     @L(@CP(88), @C(755).IN1)
    ;
  @G(1643) :
     @L(@VF(1641).o, @CP(1655)),
     @L(@CP(1655), @C(1642).G),
     @L(@CP(1655), @C(1648).G)
    ;
  @G(1647) :
     @L(@VF(1644).o, @C(1642).IN1)
    ;
  @G(1654) :
     @L(@VF(1651).o, @C(1648).IN1)
    ;
  @G(2183) :
     @L(@VF(2067).o, @C(1648).IN0)
    ;
  @G(1219) :
     @L(@CP(2193), @C(659).G),
     @L(@CP(2193), @C(2185).G),
     @L(@CP(2193), @C(543).G),
     @L(@C(672).AND, @CP(2193))
    ;
  @G(1222) :
     @L(@VF(1210).o, @C(659).IN1)
    ;
  @G(2191) :
     @L(@VF(2190).o, @C(2185).IN0)
    ;
  @G(2195) :
     @L(@VF(2192).o, @C(2185).IN1)
    ;
  @G(667) :
     @L(@C(659).SEL, @VF(665).i)
    ;
  @G(2196) :
     @L(@C(2185).SEL, @VF(2194).i)
    ;
  @G(2200) :
     @L(@C(543).SEL, @VF(684).i)
    ;
  @G(2198) :
     @L(@VF(1876).o, @C(543).IN1)
    ;
  @G(1019) :
     @L(@C(1880).DIV, @CP(1884)),
     @L(@CP(1884), @VF(1882).i),
     @L(@CP(1884), @VF(694).i)
    ;
  @G(1650) :
     @L(@C(1642).SEL, @C(1646).IN2)
    ;
  @G(2629) :
     @L(@C(1646).AND, @VF(1645).i)
    ;
  @G(2631) :
     @L(@C(1648).SEL, @C(2630).IN2)
    ;
  @G(2632) :
     @L(@C(2630).AND, @VF(1649).i)
    ;
  @G(2634) :
     @L(@VF(2633).o, @CP(2635)),
     @L(@CP(2635), @C(1646).IN1),
     @L(@CP(2635), @C(2630).IN1)
    ;
  @G(2596) :
     @L(@VF(2594).o, @CP(2606)),
     @L(@CP(2606), @C(2595).IN1),
     @L(@CP(2606), @C(2605).IN1)
    ;
  @G(2598) :
     @L(@VF(2597).o, @C(2595).IN2)
    ;
  @G(2608) :
     @L(@VF(2607).o, @C(2605).IN2)
    ;
  @G(1281) :
     @L(@VF(1277).o, @C(1278).IN1)
    ;
  @G(2600) :
     @L(@C(2595).GE, @C(2599).I)
    ;
  @G(2602) :
     @L(@VF(2601).o, @C(2599).D)
    ;
  @G(2611) :
     @L(@VF(2610).o, @C(2609).D)
    ;
  @G(2612) :
     @L(@C(2605).LE, @C(2609).I)
    ;
  @G(1276) :
     @L(@VF(1279).o, @C(1278).IN2)
    ;
  @G(1297) :
     @L(@VF(1295).o, @C(1296).IN1)
    ;
  @G(1310) :
     @L(@C(1302).Q, @C(1304).IN1)
    ;
  @G(1299) :
     @L(@VF(1298).o, @C(1296).IN2)
    ;
  @G(2604) :
     @L(@C(2599).O, @VF(2603).i)
    ;
  @G(2614) :
     @L(@C(2609).O, @VF(2613).i)
    ;
  @G(1307) :
     @L(@VF(1303).o, @C(1302).PT)
    ;
  @G(1305) :
     @L(@C(1304).OR, @C(1300).IN2)
    ;
  @G(1301) :
     @L(@C(1287).Q, @C(1304).IN2)
    ;
  @G(1288) :
     @L(@VF(1289).o, @C(1287).PT)
    ;
  @G(1275) :
     @L(@C(1300).AND, @VF(1292).i)
    ;
  @G(1343) :
     @L(@VF(1329).o, @C(1315).IN1)
    ;
  @G(2619) :
     @L(@C(2618).AND, @VF(1314).i)
    ;
  @G(1036) :
     @L(@VF(1336).o, @C(1315).IN2)
    ;
  @G(2617) :
     @L(@C(1284).Q, @C(1282).IN1)
    ;
  @G(2615) :
     @L(@VF(1311).o, @C(1283).IN1)
    ;
  @G(2621) :
     @L(@C(1282).OR, @C(2618).IN2)
    ;
  @G(1328) :
     @L(@VF(1286).o, @C(1284).PT)
    ;
  @G(2616) :
     @L(@VF(1306).o, @C(1283).IN2)
    ;
  @G(1377) :
     @L(@C(1035).Q, @C(1282).IN2)
    ;
  @G(1312) :
     @L(@VF(1285).o, @C(1035).PT)
    ;
  @G(2625) :
     @L(@VF(2622).o, @C(2624).IN1)
    ;
  @G(2628) :
     @L(@C(2624).OR, @VF(2627).i)
    ;
  @G(2626) :
     @L(@VF(2623).o, @C(2624).IN2)
    ;
  @G(1657) :
     @L(@VF(1656).o, @C(1642).IN0)
    ;
  @G(1034) :
     @L(@C(1278).OR, @CP(2366)),
     @L(@CP(1040), @C(1300).IN1),
     @L(@CP(1040), @VF(2638).i),
     @L(@CP(2366), @CP(1040)),
     @L(@CP(2366), @C(1291).IN2),
     @L(@CP(2366), @C(2358).IN2)
    ;
  @G(642) :
     @L(@C(1315).OR, @CP(2373)),
     @L(@CP(1041), @C(2618).IN1),
     @L(@CP(1041), @VF(2636).i),
     @L(@CP(2373), @CP(1041)),
     @L(@CP(2373), @C(1375).IN2),
     @L(@CP(2373), @C(1313).IN2)
    ;
  @G(373) :
     @L(@VF(585).o, @C(70).prechargeOk)
    ;
  @G(375) :
     @L(@VF(496).o, @C(70).contactFbkNeg)
    ;
  @G(376) :
     @L(@VF(1266).o, @C(70).shutdownComplete)
    ;
  @G(607) :
     @L(@VF(564).o, @C(70).chargeProtect)
    ;
  @G(683) :
     @L(@VF(617).o, @C(70).dischargeProtect)
    ;
  @G(686) :
     @L(@C(1259).LT, @VF(1264).i)
    ;
  @G(692) :
     @L(@C(70).STATE, @VF(797).i)
    ;
  @G(1043) :
     @L(@C(70).prechargeOn, @VF(1290).i)
    ;
  @G(1044) :
     @L(@C(70).contact, @VF(205).i)
    ;
  @G(1045) :
     @L(@C(70).contactNeg, @VF(999).i)
    ;
  @G(1273) :
     @L(@VF(360).o, @C(70).shutdown)
    ;
  @G(2167) :
     @L(@VF(2130).o, @C(425).IN)
    ;
  @G(500) :
     @L(@VF(520).o, @C(125).balDiff)
    ;
  @G(829) :
     @L(@VF(535).o, @C(413).Difference_Tolerance)
    ;
  @G(1047) :
     @L(@C(61).TO_USINT, @VF(17).i)
    ;
  @G(989) :
     @L(@VF(39).o, @C(1).NBOARDS)
    ;
  @G(1046) :
     @L(@VF(2310).o, @C(132).IN1)
    ;
  @G(1250) :
     @L(@VF(558).o, @C(132).IN2)
    ;
  @G(2311) :
     @L(@C(132).AND, @VF(556).i)
    ;
  @G(2246) :
     @L(@C(1779).Q, @C(1887).IN1)
    ;
  @G(2317) :
     @L(@C(42).Q, @C(1887).IN2)
    ;
  @G(2324) :
     @L(@C(2320).Q, @C(2322).IN2)
    ;
  @G(2325) :
     @L(@C(2321).Q, @C(2322).IN1)
    ;
  @G(2326) :
     @L(@VF(2236).o, @C(2624).IN3)
    ;
  @G(2335) :
     @L(@C(23).TO_UINT, @VF(610).i)
    ;
  @G(1309) :
     @L(@C(1296).GT, @C(1291).IN1)
    ;
  @G(2357) :
     @L(@C(1291).AND, @C(1302).IN)
    ;
  @G(2363) :
     @L(@C(2358).AND, @C(1287).IN)
    ;
  @G(2364) :
     @L(@VF(1293).o, @C(2358).IN1)
    ;
  @G(2367) :
     @L(@C(1283).LT, @C(1375).IN1)
    ;
  @G(2368) :
     @L(@C(1375).AND, @C(1284).IN)
    ;
  @G(2369) :
     @L(@C(1313).AND, @C(1035).IN)
    ;
  @G(2372) :
     @L(@VF(1308).o, @C(1313).IN1)
    ;
  @G(951) :
     @L(@C(146).SOC, @CP(1000)),
     @L(@CP(1000), @VF(468).i),
     @L(@CP(1000), @C(933).IN)
    ;
  @G(127) :
     @L(@C(466).Power_Counter_Wh, @VF(427).i)
    ;
  @G(416) :
     @L(@C(466).Current_mA, @VF(584).i)
    ;
  @G(343) :
     @L(@VF(69).o, @C(341).IN2)
    ;
  @G(464) :
     @L(@C(435).SEL, @VF(437).i)
    ;
  @G(561) :
     @L(@VF(560).o, @C(435).IN1)
    ;
  @G(563) :
     @L(@VF(562).o, @C(435).IN0)
    ;
  @G(566) :
     @L(@C(565).Q, @C(435).G)
    ;
  @G(568) :
     @L(@VF(567).o, @C(565).CLK)
    ;
  @G(682) :
     @L(@VF(569).o, @C(582).IN1)
    ;
  @G(740) :
     @L(@VF(739).o, @C(582).IN2)
    ;
  @G(749) :
     @L(@C(582).SUB, @C(742).IN1)
    ;
  @G(751) :
     @L(@VF(750).o, @C(742).IN2)
    ;
  @G(754) :
     @L(@C(742).GT, @C(895).R)
    ;
  @G(758) :
     @L(@VF(1743).o, @C(757).IN2)
    ;
  @G(855) :
     @L(@VF(1730).o, @C(757).IN1)
    ;
  @G(857) :
     @L(@C(757).GE, @C(1702).IN2)
    ;
  @G(894) :
     @L(@VF(889).o, @C(861).IN0)
    ;
  @G(896) :
     @L(@VF(886).o, @C(861).IN1)
    ;
  @G(898) :
     @L(@C(866).Q, @C(861).G)
    ;
  @G(901) :
     @L(@VF(890).o, @C(866).CLK)
    ;
  @G(892) :
     @L(@C(861).SEL, @VF(867).i)
    ;
  @G(1021) :
     @L(@VF(952).o, @C(926).IN2)
    ;
  @G(1022) :
     @L(@C(944).SUB, @C(926).IN1)
    ;
  @G(1023) :
     @L(@VF(987).o, @C(944).IN1)
    ;
  @G(1030) :
     @L(@VF(1020).o, @C(944).IN2)
    ;
  @G(1033) :
     @L(@C(926).GT, @C(329).R)
    ;
  @G(347) :
     @L(@C(1).MINTEMP, @VF(346).i)
    ;
  @G(1084) :
     @L(@C(1).MAXTEMP, @VF(344).i)
    ;
  @G(130) :
     @L(@C(854).O, @C(878).S1)
    ;
  @G(89) :
     @L(@C(858).O, @C(878).R)
    ;
  @G(92) :
     @L(@C(90).cmd0, @C(91).IN0)
    ;
  @G(93) :
     @L(@C(90).cmd1, @C(91).IN1)
    ;
  @G(95) :
     @L(@C(90).cmd2, @C(91).IN2)
    ;
  @G(345) :
     @L(@C(90).cmd3, @C(91).IN3)
    ;
  @G(378) :
     @L(@C(91).MUX_USINT, @VF(355).i)
    ;
  @G(381) :
     @L(@VF(380).o, @CP(382)),
     @L(@CP(382), @C(2255).K),
     @L(@CP(382), @C(91).K)
    ;
  @G(385) :
     @L(@VF(383).o, @C(384).IN1)
    ;
  @G(387) :
     @L(@VF(386).o, @C(384).IN2)
    ;
  @G(851) :
     @L(@C(384).EQ, @VF(619).i)
    ;
  @G(1129) :
     @L(@VF(864).o, @C(859).IN2)
    ;
  @G(1135) :
     @L(@VF(1091).o, @C(859).IN1)
    ;
  @G(1138) :
     @L(@C(859).EQ, @VF(1115).i)
    ;
  @G(1144) :
     @L(@VF(1140).o, @C(1139).IN2)
    ;
  @G(1145) :
     @L(@VF(1142).o, @C(1139).IN1)
    ;
  @G(1146) :
     @L(@C(1139).EQ, @VF(1143).i)
    ;
  @G(669) :
     @L(@VF(1203).o, @C(657).IN1)
    ;
  @G(670) :
     @L(@VF(1204).o, @C(657).IN2)
    ;
  @G(671) :
     @L(@VF(2265).o, @C(90).CAN_ID)
    ;
  @G(1149) :
     @L(@C(90).CAN_Error, @VF(1148).i)
    ;
  @G(673) :
     @L(@C(657).GT, @C(672).IN2)
    ;
  @G(1157) :
     @L(@VF(1150).o, @C(672).IN1)
    ;
  @G(748) :
     @L(@VF(812).o, @C(699).temp)
    ;
  @G(775) :
     @L(@C(699).mult, @C(838).IN1)
    ;
  @G(828) :
     @L(@VF(819).o, @C(817).temp)
    ;
  @G(1008) :
     @L(@C(817).mult, @C(838).IN2)
    ;
  @G(1068) :
     @L(@VF(1077).o, @C(1014).temp)
    ;
  @G(1173) :
     @L(@C(1014).mult, @C(1195).IN1)
    ;
  @G(1193) :
     @L(@VF(1191).o, @C(1192).temp)
    ;
  @G(1196) :
     @L(@C(1192).mult, @C(1195).IN2)
    ;
  @G(1202) :
     @L(@C(1195).MIN, @C(1201).IN1)
    ;
  @G(1205) :
     @L(@C(1198).mult, @C(1201).IN2)
    ;
  @G(1206) :
     @L(@C(1201).MUL, @VF(1200).i)
    ;
  @G(1208) :
     @L(@C(1016).MUL, @VF(690).i)
    ;
  @G(1234) :
     @L(@VF(1231).o, @C(1207).maxCell)
    ;
  @G(1236) :
     @L(@VF(1235).o, @C(1198).minCell)
    ;
  @G(1246) :
     @L(@VF(1240).o, @C(1207).chargeOn)
    ;
  @G(1248) :
     @L(@VF(1247).o, @C(1198).discOn)
    ;
  @G(644) :
     @L(@VF(357).o, @C(303).IN1)
    ;
  @G(656) :
     @L(@VF(379).o, @C(303).IN2)
    ;
  @G(796) :
     @L(@VF(555).o, @C(302).PT)
    ;
  @G(798) :
     @L(@C(303).EQ, @C(302).IN)
    ;
  @G(865) :
     @L(@C(302).Q, @VF(831).i)
    ;
  @G(930) :
     @L(@VF(905).o, @C(874).IN1)
    ;
  @G(931) :
     @L(@VF(909).o, @C(874).IN2)
    ;
  @G(942) :
     @L(@C(874).GE, @C(904).IN1)
    ;
  @G(945) :
     @L(@VF(923).o, @C(904).IN2)
    ;
  @G(1249) :
     @L(@C(904).AND, @VF(198).i)
    ;
  @G(1316) :
     @L(@VF(1280).o, @C(1274).IN2)
    ;
  @G(1317) :
     @L(@VF(1294).o, @C(1274).IN1)
    ;
  @G(1363) :
     @L(@VF(1267).o, @C(1319).IN1)
    ;
  @G(1396) :
     @L(@VF(1318).o, @C(1319).IN2)
    ;
  @G(1462) :
     @L(@VF(1461).o, @C(1450).IN2)
    ;
  @G(1553) :
     @L(@VF(1453).o, @C(1450).IN1)
    ;
  @G(1652) :
     @L(@C(1319).LE, @C(1640).IN1)
    ;
  @G(1707) :
     @L(@VF(1653).o, @C(1640).IN2)
    ;
  @G(1740) :
     @L(@C(1640).AND, @C(1709).IN3)
    ;
  @G(1741) :
     @L(@C(1450).OR, @C(1709).IN2)
    ;
  @G(1742) :
     @L(@C(1274).LT, @C(1709).IN1)
    ;
  @G(1744) :
     @L(@C(1709).OR, @VF(1252).i)
    ;
  @G(735) :
     @L(@VF(625).o, @CP(738)),
     @L(@CP(738), @C(2321).CLK),
     @L(@CP(738), @C(2320).CLK)
    ;
  @G(1764) :
     @L(@C(1790).SEL, @VF(1829).i)
    ;
  @G(1774) :
     @L(@VF(1769).o, @C(1790).G)
    ;
  @G(1768) :
     @L(@C(1780).TO_REAL, @C(1783).IN1)
    ;
  @G(1793) :
     @L(@VF(1765).o, @C(1783).IN2)
    ;
  @G(1801) :
     @L(@VF(1798).o, @C(1795).IN1)
    ;
  @G(1808) :
     @L(@VF(1797).o, @C(1795).IN2)
    ;
  @G(1843) :
     @L(@C(1795).EQ, @C(1796).IN)
    ;
  @G(1844) :
     @L(@VF(1800).o, @C(1796).PT)
    ;
  @G(1845) :
     @L(@C(1796).Q, @VF(1794).i)
    ;
  @G(1858) :
     @L(@VF(1854).o, @C(1847).IN1)
    ;
  @G(1859) :
     @L(@VF(1853).o, @C(1847).IN2)
    ;
  @G(1865) :
     @L(@C(1847).LE, @C(1864).IN1)
    ;
  @G(1873) :
     @L(@VF(1867).o, @C(1864).IN2)
    ;
  @G(1946) :
     @L(@VF(1891).o, @C(1864).IN3)
    ;
  @G(1949) :
     @L(@C(1864).AND, @VF(1855).i)
    ;
  @G(2029) :
     @L(@VF(2027).o, @C(2028).IN1)
    ;
  @G(2089) :
     @L(@VF(2026).o, @C(2028).IN2)
    ;
  @G(2099) :
     @L(@VF(2097).o, @C(2092).IN1)
    ;
  @G(2100) :
     @L(@VF(2098).o, @C(2092).IN2)
    ;
  @G(2102) :
     @L(@C(2092).GT, @C(2101).IN1)
    ;
  @G(2104) :
     @L(@C(2028).GE, @C(2103).IN1)
    ;
  @G(2106) :
     @L(@VF(2105).o, @C(2103).IN2)
    ;
  @G(2108) :
     @L(@VF(2107).o, @C(2103).IN3)
    ;
  @G(2109) :
     @L(@C(2103).AND, @C(2101).IN2)
    ;
  @G(2113) :
     @L(@VF(2111).o, @C(2110).IN2)
    ;
  @G(2114) :
     @L(@VF(2112).o, @C(2110).IN1)
    ;
  @G(2115) :
     @L(@C(2110).OR, @C(2101).IN3)
    ;
  @G(2118) :
     @L(@C(2101).OR, @VF(2117).i)
    ;
  @G(2091) :
     @L(@C(1787).SEL, @VF(1816).i)
    ;
  @G(626) :
     @L(@VF(356).o, @C(1770).IN2)
    ;
  @G(1791) :
     @L(@C(1781).TO_REAL, @C(1782).IN1)
    ;
  @G(1804) :
     @L(@VF(1803).o, @C(1782).IN2)
    ;
  @G(1809) :
     @L(@VF(1807).o, @CP(1811)),
     @L(@CP(1811), @C(1779).CLK),
     @L(@CP(1811), @C(42).CLK)
    ;
  @G(1828) :
     @L(@VF(1812).o, @C(1787).G)
    ;
  @G(1833) :
     @L(@C(64).MAX, @C(1790).IN1)
    ;
  @G(1786) :
     @L(@C(1783).MUL, @C(64).IN2)
    ;
  @G(1784) :
     @L(@VF(1810).o, @CP(1846)),
     @L(@CP(1846), @C(1790).IN0),
     @L(@CP(1846), @C(64).IN1)
    ;
  @G(1849) :
     @L(@C(1782).MUL, @C(1848).IN2)
    ;
  @G(1850) :
     @L(@C(1848).MAX, @C(1787).IN1)
    ;
  @G(1852) :
     @L(@VF(2355).o, @CP(1866)),
     @L(@CP(1866), @C(1787).IN0),
     @L(@CP(1866), @C(1848).IN1)
    ;
  @G(1875) :
     @L(@VF(1874).o, @C(1872).IN1)
    ;
  @G(1879) :
     @L(@VF(1869).o, @C(1872).IN2)
    ;
  @G(1881) :
     @L(@C(1872).MUL, @VF(1841).i)
    ;
  @G(1890) :
     @L(@VF(1888).o, @C(1889).IN1)
    ;
  @G(1893) :
     @L(@VF(1892).o, @C(1889).IN2)
    ;
  @G(1895) :
     @L(@C(1889).MUL, @VF(1894).i)
    ;
  @G(1211) :
     @L(@C(838).MIN, @C(1016).IN1)
    ;
  @G(1217) :
     @L(@C(1207).mult, @C(1016).IN2)
    ;
  @G(1766) :
     @L(@VF(63).o, @C(1770).IN1)
    ;
  @G(1792) :
     @L(@VF(1760).o, @C(1762).IN1)
    ;
  @G(1763) :
     @L(@VF(873).o, @C(1759).CU)
    ;
  @G(1773) :
     @L(@VF(1761).o, @C(1759).CD)
    ;
  @G(1777) :
     @L(@VF(1805).o, @C(1759).uPer)
    ;
  @G(1857) :
     @L(@VF(1806).o, @C(1759).dPer)
    ;
  @G(1862) :
     @L(@C(1771).TO_INT, @C(1759).PV)
    ;
  @G(1870) :
     @L(@C(2322).OR, @C(1759).RST)
    ;
  @G(1871) :
     @L(@C(1759).CV, @C(1780).IN)
    ;
  @G(1785) :
     @L(@VF(1778).o, @C(1776).CU)
    ;
  @G(1878) :
     @L(@VF(1775).o, @C(1776).CD)
    ;
  @G(1883) :
     @L(@VF(2348).o, @C(1776).uPer)
    ;
  @G(1886) :
     @L(@VF(2349).o, @C(1776).dPer)
    ;
  @G(1896) :
     @L(@C(1772).TO_INT, @C(1776).PV)
    ;
  @G(1898) :
     @L(@C(1887).OR, @C(1776).RST)
    ;
  @G(2093) :
     @L(@C(1776).CV, @C(1781).IN)
    ;
  @G(641) :
     @L(@VF(220).o, @C(83).CAN_ID)
    ;
  @G(734) :
     @L(@VF(202).o, @C(83).Max_Temp_Cell_Loc)
    ;
  @G(843) :
     @L(@VF(203).o, @C(83).Max_Temp_BMU_Loc)
    ;
  @G(1162) :
     @L(@VF(204).o, @C(83).Min_Temp_Cell_Loc)
    ;
  @G(1163) :
     @L(@VF(215).o, @C(83).Min_Temp_BMU_Loc)
    ;
  @G(1164) :
     @L(@VF(216).o, @C(83).Max_Cell_Temp)
    ;
  @G(1165) :
     @L(@VF(219).o, @C(83).Min_Cell_Temp)
    ;
  @G(221) :
     @L(@VF(518).o, @C(83).outVolt)
    ;
  @G(308) :
     @L(@VF(122).o, @C(136).CAN_ID)
    ;
  @G(397) :
     @L(@VF(143).o, @C(136).State)
    ;
  @G(408) :
     @L(@VF(1751).o, @C(136).Contactor_Status)
    ;
  @G(409) :
     @L(@VF(1131).o, @C(136).ChargeContact)
    ;
  @G(411) :
     @L(@VF(85).o, @C(136).DMDC)
    ;
  @G(412) :
     @L(@VF(87).o, @C(136).DMCC)
    ;
  @G(428) :
     @L(@VF(1130).o, @C(136).NegContact)
    ;
  @G(429) :
     @L(@VF(991).o, @C(136).isolationStatus)
    ;
  @G(434) :
     @L(@VF(238).o, @C(136).chargeComplete)
    ;
  @G(442) :
     @L(@VF(178).o, @C(136).dischargeComplete)
    ;
  @G(475) :
     @L(@VF(241).o, @C(136).in1Status)
    ;
  @G(481) :
     @L(@VF(242).o, @C(136).in2Status)
    ;
  @G(116) :
     @L(@C(84).CAN_Error, @VF(780).i)
    ;
  @G(134) :
     @L(@C(83).CAN_Error, @VF(746).i)
    ;
  @G(444) :
     @L(@VF(441).o, @C(84).CAN_ID)
    ;
  @G(480) :
     @L(@VF(244).o, @C(84).SoC)
    ;
  @G(689) :
     @L(@VF(260).o, @C(84).SoH)
    ;
  @G(695) :
     @L(@VF(990).o, @C(84).Duty_Cycle)
    ;
  @G(696) :
     @L(@VF(58).o, @C(84).Available_Energy)
    ;
  @G(697) :
     @L(@VF(133).o, @C(84).Remain_Energy)
    ;
  @G(1168) :
     @L(@VF(983).o, @C(700).R)
    ;
  @G(1170) :
     @L(@VF(1167).o, @C(700).CODE)
    ;
  @G(1171) :
     @L(@C(700).VAL, @C(733).IN)
    ;
  @G(1175) :
     @L(@C(733).TO_UDINT, @C(1172).IN)
    ;
  @G(1364) :
     @L(@C(1172).TO_TIME, @C(1176).IN1)
    ;
  @G(1365) :
     @L(@C(1176).DIV_TIME, @VF(1166).i)
    ;
  @G(1369) :
     @L(@VF(1366).o, @C(1176).IN2)
    ;
  @G(1928) :
     @L(@VF(1385).o, @C(1372).PT)
    ;
  @G(1929) :
     @L(@VF(1384).o, @C(1371).PT)
    ;
  @G(1930) :
     @L(@C(1371).Q, @VF(1386).i)
    ;
  @G(1931) :
     @L(@C(1372).Q, @CP(1926)),
     @L(@CP(1926), @C(1371).IN),
     @L(@CP(1926), @VF(1382).i),
     @L(@CP(1926), @VF(1383).i)
    ;
  @G(1932) :
     @L(@VF(1387).o, @C(1372).IN)
    ;
  @G(1933) :
     @L(@VF(1392).o, @C(1378).CH)
    ;
  @G(1934) :
     @L(@C(1374).OUT, @C(1373).VAL)
    ;
  @G(1935) :
     @L(@VF(1638).o, @C(1373).PIN)
    ;
  @G(1936) :
     @L(@VF(1917).o, @C(1373).PORT)
    ;
  @G(1937) :
     @L(@VF(1639).o, @C(1379).IN2)
    ;
  @G(1938) :
     @L(@VF(1916).o, @C(1378).GRP)
    ;
  @G(1939) :
     @L(@VF(1393).o, @C(1380).PT)
    ;
  @G(1940) :
     @L(@VF(1915).o, @C(1381).PT)
    ;
  @G(1941) :
     @L(@VF(1918).o, @C(1374).PER)
    ;
  @G(1947) :
     @L(@VF(1921).o, @C(1374).IN)
    ;
  @G(1948) :
     @L(@VF(1922).o, @C(1376).SLEEP_RDY)
    ;
  @G(1952) :
     @L(@C(1380).Q, @C(1381).IN)
    ;
  @G(1953) :
     @L(@C(1379).GT, @C(1380).IN)
    ;
  @G(1954) :
     @L(@C(1378).VAL, @CP(1927)),
     @L(@CP(1927), @C(1379).IN1),
     @L(@CP(1927), @VF(1923).i)
    ;
  @G(1955) :
     @L(@C(1381).Q, @VF(1920).i)
    ;
  @G(1956) :
     @L(@VF(1919).o, @C(1378).ADC)
    ;
  @G(2150) :
     @L(@VF(1968).o, @C(1957).IN1)
    ;
  @G(2151) :
     @L(@VF(1967).o, @C(1957).IN2)
    ;
  @G(2163) :
     @L(@C(1957).EQ, @C(1958).G)
    ;
  @G(2164) :
     @L(@VF(1970).o, @C(1958).IN0)
    ;
  @G(2165) :
     @L(@VF(1969).o, @C(1958).IN1)
    ;
  @G(2169) :
     @L(@VF(1971).o, @C(1959).PORT)
    ;
  @G(2170) :
     @L(@VF(1972).o, @C(1959).PIN)
    ;
  @G(2171) :
     @L(@C(1958).SEL, @C(1959).VAL)
    ;
  @G(2172) :
     @L(@VF(1975).o, @C(1961).VAL)
    ;
  @G(2182) :
     @L(@VF(1974).o, @C(1961).PIN)
    ;
  @G(2184) :
     @L(@VF(1973).o, @C(1961).PORT)
    ;
  @G(2186) :
     @L(@VF(1976).o, @C(1960).PORT)
    ;
  @G(2187) :
     @L(@VF(2008).o, @C(1960).PIN)
    ;
  @G(2188) :
     @L(@VF(2009).o, @C(1960).VAL)
    ;
  @G(2189) :
     @L(@VF(2119).o, @C(1962).PORT)
    ;
  @G(2210) :
     @L(@VF(2120).o, @C(1962).PIN)
    ;
  @G(2211) :
     @L(@VF(2121).o, @C(1962).VAL)
    ;
  @G(2215) :
     @L(@VF(2122).o, @C(1964).PORT)
    ;
  @G(2216) :
     @L(@VF(2123).o, @C(1964).PIN)
    ;
  @G(2217) :
     @L(@VF(2124).o, @C(1964).VAL)
    ;
  @G(2218) :
     @L(@VF(2125).o, @C(1965).PORT)
    ;
  @G(2219) :
     @L(@VF(2126).o, @C(1965).PIN)
    ;
  @G(2220) :
     @L(@VF(2127).o, @C(1966).IN)
    ;
  @G(2221) :
     @L(@C(1966).OUT, @C(1965).VAL)
    ;
  @G(2222) :
     @L(@VF(2128).o, @C(1966).PER)
    ;
  @G(2268) :
     @L(@VF(2231).o, @C(2225).PIN)
    ;
  @G(2270) :
     @L(@VF(2240).o, @C(2223).PORT)
    ;
  @G(2272) :
     @L(@VF(2229).o, @C(2223).PIN)
    ;
  @G(2278) :
     @L(@VF(2238).o, @C(2224).PORT)
    ;
  @G(2280) :
     @L(@VF(2230).o, @C(2224).PIN)
    ;
  @G(2281) :
     @L(@VF(2239).o, @C(2225).PORT)
    ;
  @G(2282) :
     @L(@VF(2232).o, @C(2226).PIN)
    ;
  @G(2283) :
     @L(@VF(2235).o, @C(2226).PORT)
    ;
  @G(2284) :
     @L(@VF(2233).o, @C(2227).PIN)
    ;
  @G(2285) :
     @L(@VF(2241).o, @C(2227).PORT)
    ;
  @G(2289) :
     @L(@VF(2234).o, @C(2228).PIN)
    ;
  @G(2290) :
     @L(@VF(2249).o, @C(2228).PORT)
    ;
  @G(1012) :
     @L(@VF(487).o, @C(452).CH)
    ;
  @G(1013) :
     @L(@VF(491).o, @C(471).CH)
    ;
  @G(1015) :
     @L(@VF(707).o, @C(240).CH)
    ;
  @G(1017) :
     @L(@VF(1444).o, @C(200).CH)
    ;
  @G(2305) :
     @L(@VF(1439).o, @C(1361).ch)
    ;
  @G(2306) :
     @L(@VF(1398).o, @C(1350).ch)
    ;
  @G(2307) :
     @L(@VF(1440).o, @C(1362).ch)
    ;
  @G(2308) :
     @L(@VF(1442).o, @C(1341).PORT)
    ;
  @G(2309) :
     @L(@VF(1443).o, @C(1341).PIN)
    ;
  @G(2312) :
     @L(@VF(2287).o, @C(1340).PIN)
    ;
  @G(2314) :
     @L(@VF(2264).o, @C(1340).PORT)
    ;
  @G(2315) :
     @L(@VF(2291).o, @C(1018).PORT)
    ;
  @G(2316) :
     @L(@VF(2292).o, @C(1018).PIN)
    ;
  @G(2318) :
     @L(@VF(2293).o, @C(1388).PORT)
    ;
  @G(2319) :
     @L(@VF(2294).o, @C(1388).PIN)
    ;
  @G(2323) :
     @L(@VF(2295).o, @C(1397).PORT)
    ;
  @G(2328) :
     @L(@VF(2296).o, @C(1397).PIN)
    ;
  @G(59) :
     @L(@VF(1438).o, @C(452).GRP)
    ;
  @G(112) :
     @L(@VF(705).o, @C(452).ADC)
    ;
  @G(152) :
     @L(@VF(139).o, @C(471).ADC)
    ;
  @G(153) :
     @L(@VF(140).o, @C(471).GRP)
    ;
  @G(169) :
     @L(@VF(145).o, @C(240).ADC)
    ;
  @G(193) :
     @L(@VF(147).o, @C(240).GRP)
    ;
  @G(212) :
     @L(@VF(148).o, @C(200).ADC)
    ;
  @G(214) :
     @L(@VF(150).o, @C(200).GRP)
    ;
  @G(224) :
     @L(@C(223).OR, @C(146).memoryWrite)
    ;
  @G(225) :
     @L(@C(815).Q, @C(223).IN1)
    ;
  @G(230) :
     @L(@C(226).Q, @C(223).IN2)
    ;
  @G(233) :
     @L(@VF(232).o, @C(226).CLK)
    ;
  @G(1522) :
     @L(@C(1427).TEMP, @VF(1467).i)
    ;
  @G(1518) :
     @L(@VF(1458).o, @C(1427).VSUP)
    ;
  @G(1517) :
     @L(@VF(1457).o, @C(1427).RS)
    ;
  @G(1514) :
     @L(@VF(1459).o, @C(1427).BETA)
    ;
  @G(1515) :
     @L(@VF(1456).o, @C(1427).TNOM)
    ;
  @G(1516) :
     @L(@VF(1460).o, @C(1427).RNOM)
    ;
  @G(704) :
     @L(@VF(820).o, @VF(2135).i)
    ;
  @G(719) :
     @L(@VF(469).o, @VF(149).i)
    ;
  @G(47) :
     @L(@VF(525).o, @C(43).IN1)
    ;
  @G(760) :
     @L(@VF(448).o, @VF(759).i)
    ;
  @G(761) :
     @L(@VF(239).o, @VF(756).i)
    ;
  @G(771) :
     @L(@C(43).DIV, @VF(747).i)
    ;
  @G(846) :
     @L(@VF(844).o, @C(833).IN2)
    ;
  @G(847) :
     @L(@VF(837).o, @C(833).IN1)
    ;
  @G(849) :
     @L(@C(833).OR, @VF(834).i)
    ;
  @G(947) :
     @L(@C(1002).TO_USINT, @C(763).PV)
    ;
  @G(1005) :
     @L(@VF(853).o, @C(1002).IN)
    ;
  @G(1064) :
     @L(@VF(1063).o, @C(804).MaxBMU)
    ;
  @G(1065) :
     @L(@VF(1010).o, @C(804).indx)
    ;
  @G(1066) :
     @L(@VF(1009).o, @C(804).Map)
    ;
  @G(1067) :
     @L(@VF(1007).o, @C(804).CellCounter)
    ;
  @G(1069) :
     @L(@C(804).Reset, @VF(1062).i)
    ;
  @G(1070) :
     @L(@C(804).numofCell, @VF(1011).i)
    ;
  @G(744) :
     @L(@VF(231).o, @C(762).R)
    ;
  @G(363) :
     @L(@VF(359).o, @C(70).contactFbk)
    ;
  @G(3262) :
     @L(@VF(3239).o, @CP(776)),
     @L(@CP(776), @C(3226).ENB),
     @L(@CP(776), @C(1083).IN1)
    ;
  @G(3261) :
     @L(@VF(3241).o, @C(3226).CAN_CH)
    ;
  @G(3269) :
     @L(@C(3226).CANerr, @VF(3249).i)
    ;
  @G(3264) :
     @L(@VF(3242).o, @C(3224).IN)
    ;
  @G(3270) :
     @L(@C(3231).SUB, @C(3229).IN)
    ;
  @G(3272) :
     @L(@CP(3256), @C(3231).IN1),
     @L(@CP(3256), @C(3228).IN1),
     @L(@VF(3245).o, @CP(3256))
    ;
  @G(3263) :
     @L(@C(3224).TO_TIME, @C(3225).IN1)
    ;
  @G(3265) :
     @L(@VF(3243).o, @C(3225).IN2)
    ;
  @G(3267) :
     @L(@VF(3244).o, @C(3228).IN2)
    ;
  @G(3271) :
     @L(@C(3229).ABS, @C(3232).IN1)
    ;
  @G(3275) :
     @L(@VF(3247).o, @C(3232).IN2)
    ;
  @G(3276) :
     @L(@VF(3246).o, @C(3231).IN2)
    ;
  @G(3277) :
     @L(@CP(3257), @C(3230).PT),
     @L(@CP(3257), @C(3238).PT),
     @L(@C(3225).DIV_TIME, @CP(3257))
    ;
  @G(3273) :
     @L(@C(3232).LT, @C(3230).IN)
    ;
  @G(3280) :
     @L(@VF(3250).o, @C(3233).IN2)
    ;
  @G(3281) :
     @L(@CP(3258), @C(3236).IN1),
     @L(@CP(3258), @C(3233).IN1),
     @L(@VF(3252).o, @CP(3258))
    ;
  @G(3282) :
     @L(@C(3236).SUB, @C(3235).IN)
    ;
  @G(3283) :
     @L(@C(3235).ABS, @C(3237).IN1)
    ;
  @G(3284) :
     @L(@C(3237).LT, @C(3238).IN)
    ;
  @G(3266) :
     @L(@C(3228).GT, @C(3227).IN1)
    ;
  @G(3274) :
     @L(@C(3230).Q, @C(3227).IN2)
    ;
  @G(3278) :
     @L(@C(3233).GT, @C(3234).IN1)
    ;
  @G(3285) :
     @L(@C(3238).Q, @C(3234).IN2)
    ;
  @G(3286) :
     @L(@VF(3254).o, @C(3236).IN2)
    ;
  @G(3287) :
     @L(@VF(3253).o, @C(3237).IN2)
    ;
  @G(3268) :
     @L(@C(3227).AND, @VF(3248).i)
    ;
  @G(3279) :
     @L(@C(3234).AND, @VF(3251).i)
    ;
  @G(358) :
     @L(@VF(621).o, @C(70).discharge)
    ;
  @G(374) :
     @L(@VF(1323).o, @C(70).charge)
    ;
  @G(253) :
     @L(@VF(237).o, @C(2228).VAL)
    ;
  @G(453) :
     @L(@VF(236).o, @C(2227).VAL)
    ;
  @G(330) :
     @L(@VF(310).o, @CP(436)),
     @L(@CP(436), @C(850).IN1),
     @L(@CP(436), @C(175).IN2)
    ;
  @G(703) :
     @L(@C(1361).stat, @C(175).IN1)
    ;
  @G(721) :
     @L(@C(1362).stat, @C(850).IN2)
    ;
  @G(731) :
     @L(@C(850).EQ, @VF(722).i)
    ;
  @G(741) :
     @L(@C(175).EQ, @VF(723).i)
    ;
  @G(810) :
     @L(@VF(196).o, @C(543).IN0)
    ;
  @G(1006) :
     @L(@VF(811).o, @C(908).IN1)
    ;
  @G(1072) :
     @L(@VF(821).o, @C(908).IN2)
    ;
  @G(1075) :
     @L(@C(908).OR, @VF(1074).i)
    ;
  @G(668) :
     @L(@VF(662).o, @C(659).IN0)
    ;
  @G(557) :
     @L(@VF(195).o, @C(70).fault)
    ;
  @G(449) :
     @L(@VF(1076).o, @C(136).emergencyButton)
    ;
  @G(1085) :
     @L(@C(1083).AND, @C(3226).RST)
    ;
  @G(1087) :
     @L(@VF(1086).o, @C(1083).IN2)
    ;
  @G(1078) :
     @L(@VF(1963).o, @VF(1003).i)
    ;
  @G(22) :
     @L(@VF(1476).o, @C(14).CODE)
    ;
  @G(688) :
     @L(@VF(1528).o, @C(14).R)
    ;
  @G(1080) :
     @L(@C(14).VAL, @C(1079).IN)
    ;
  @G(1081) :
     @L(@C(1079).TO_USINT, @VF(581).i)
    ;
  @G(489) :
     @L(@C(452).VAL, @C(1427).VOLT)
    ;
  @G(474) :
     @L(@VF(410).o, @C(136).Ambient_Temp)
    ;
END_PROGRAM
